TYPE ST_PickPlaceArmConfig :
STRUCT

END_STRUCT
END_TYPE

(* stored: Version 1.1.0.1, ProductVersion 3.1.4024.9
   DUT ST_PickPlaceArmConfig: Id {9c0230be-080f-4ca8-b2d1-76be4dc4fe1b} *)
